// Mitsubishi GX Works2 project: 断电延时动作的程序   PLC: FX2N/FX2NC

PROGRAM MAIN
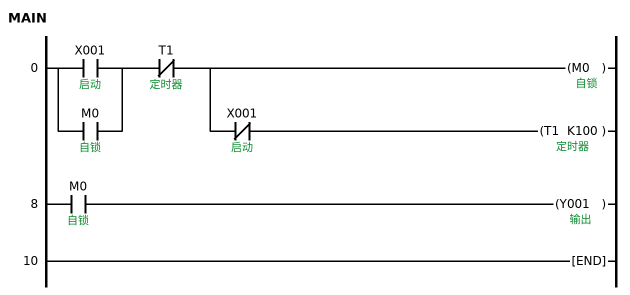
; 
0     LD      X001  ; 启动
      OR      M0  ; 自锁
      ANI     T1  ; 定时器
      OUT     M0  ; 自锁
      ANI     X001  ; 启动
      OUT     T1 K100  ; 定时器
8     LD      M0  ; 自锁
      OUT     Y001  ; 输出
10    END
END_PROGRAM
